// TIA Portal V21 export
TYPE "LAxisCtrl_typeStop"
TITLE = LAxisCtrl_typeStop
// Support: tech.team.motioncontrol@siemens.com
   STRUCT
      deceleration : LReal := -1.0;   // Deceleration setpoint for stop (Value > 0.0: The specified value is used; Value = 0.0: Not permitted; Value < 0.0: Use of the default value configured in the technology object)
      jerk : LReal := -1.0;   // Jerk for stop (Value > 0.0: Smooth velocity profile, the specified value is used; Value = 0.0: Trapezoid velocity profile; Value < 0.0: Use of the default value configured in the technology object)
      abortAcceleration : Bool := FALSE;   // TRUE: The acceleration is set to 0.0 at the start of the job, and the deceleration immediately builds up; FALSE: The current acceleration at the start of the job is reduced using the configured jerk. Afterwards, the deceleration builds up
      haltMode : DInt := 0;   // Select the motion which is to be stopped (0: The basic motion and the superimposed motion are stopped; 1: The basic motion is stopped. The superimposed motion remains active)
   END_STRUCT;
END_TYPE
